// TIA Portal V17 export
// export: Created 2025-03-10T12:16:58.0432232Z, ExportSetting WithDefaults, DisplayName Totally Integrated Automation Portal, DisplayVersion V17 Update 8, DisplayName TIA Portal Openness, DisplayVersion V17 Update 8, DisplayName TIA Portal Version Control Interface, DisplayVersion V17, DisplayName SINAMICS Startdrive Advanced, DisplayVersion V17 SP2, DisplayName SINAMICS Startdrive G110M, G120, G120C, G120D, G120P, G115D, DisplayVersion V17 SP2, DisplayName SINAMICS Startdrive G130, G150, S120, S150, SINAMICS MV, S210, DisplayVersion V17 SP2, DisplayName STEP 7 Professional, DisplayVersion V17 Update 8, DisplayName SINUMERIK ONE STEP 7 Toolbox, DisplayVersion V17 Update 12, DisplayName SINUMERIK 840D sl STEP 7 Toolbox, DisplayVersion V17 Update 12, DisplayName STEP 7 Safety, DisplayVersion V17 Update 6, DisplayName WinCC Advanced, DisplayVersion V17 Update 8
DATA_BLOCK "DB6890_UNIT_02_STA_3_ANGULAR_LOCATOR"   // DB6890
{ DB_Accessible_From_OPC_UA := 'FALSE' }
AUTHOR : ETXETAR
VERSION : 1.0
// stored: AutoNumber false, DBAccessibleFromOPCUA false, DBAccessibleFromWebserver true, InstanceOfName FB6500_CYLINDER, InstanceOfType FB
"FB6500_CYLINDER"
   // VAR_INPUT
   //    OPTIONS_0 : Byte;
   //    ADVANCED_1_I : Bool;
   //    ADVANCED_2_I : Bool;
   //    ADVANCED_3_I : Bool;
   //    ADVANCED_4_I : Bool;
   //    RETURNED_1_I : Bool;
   //    RETURNED_2_I : Bool;
   //    RETURNED_3_I : Bool;
   //    RETURNED_4_I : Bool;
   //    ADVANCE_CONDITIONS : Bool;
   //    RETURN_CONDITIONS : Bool;
   //    HMI_LINE_REQUEST : Bool;
   //    ADVANCE_AUTO_REQUEST : Bool;
   //    RETURN_AUTO_REQUEST : Bool;
   //    UNIT_ALARM : UInt;
   //    STATION_ALARM : UInt;
   // END_VAR
   // VAR_OUTPUT
   //    ADVANCED : Bool;
   //    RETURNED : Bool;
   //    ADVANCED_1_ALARM : Bool;
   //    ADVANCED_2_ALARM : Bool;
   //    ADVANCED_3_ALARM : Bool;
   //    ADVANCED_4_ALARM : Bool;
   //    RETURNED_1_ALARM : Bool;
   //    RETURNED_2_ALARM : Bool;
   //    RETURNED_3_ALARM : Bool;
   //    RETURNED_4_ALARM : Bool;
   //    HMI_MOTION_EXECUTABILITY_LEFT : Bool;
   //    HMI_MOTION_EXECUTABILITY_RIGHT : Bool;
   //    HMI_MOTION_END_POS_LEFT : Bool;
   //    HMI_MOTION_END_POS_RIGHT : Bool;
   //    HMI_MOTION_ACTIVE_LEFT : Bool;
   //    HMI_MOTION_ACTIVE_RIGHT : Bool;
   //    ADVANCE : Bool;
   //    "RETURN" : Bool;
   // END_VAR
   // VAR RETAIN
   //    CYL { S7_SetPoint := 'True'} : "ADVANCE_RETURN_CYL_CLADDING";
   //    TIMER_ADVANCED { S7_SetPoint := 'True'} : TON_TIME;
   //    TIMER_RETURNED { S7_SetPoint := 'True'} : TON_TIME;
   //    TIMER_SIMULTANEITY { S7_SetPoint := 'True'} : TON_TIME;
   //    TIMER_TIME_EXCEEDED { S7_SetPoint := 'True'} : TON_TIME;
   // END_VAR
BEGIN
END_DATA_BLOCK
